// Mitsubishi GX Works2 project: PLC_Group_12   PLC: FX3G

// global labels: Global1
VAR_GLOBAL CONSTANT
  Mixing_Premium_Time : INT := 50;
END_VAR
VAR_GLOBAL
  StartDay AT X007 : BOOL;
  EmergencyStop AT X005 : BOOL;
  LackOfMaterial AT M1 : BOOL;
  DayActive AT M0 : BOOL;
  WorkdayLamp AT Y007 : BOOL;
  RaspberryStock AT D1200 : REAL;
  LemonStock AT D1210 : REAL;
  InitLemon AT D1110 : REAL;
  InitStabilizer AT D1120 : REAL;
  StabilizerStock AT D1220 : REAL;
  BearsStock AT D1230 : REAL;
  InitBears AT D1130 : REAL;
  StorageCount AT D1300 : REAL;
  AnalogOutput AT D8282 : INT;
  StartPreparation AT X001 : BOOL;
  IsPremium AT M3 : BOOL;
  AnalogInput1 AT D8280 : INT;
END_VAR
VAR_GLOBAL CONSTANT
  MinRaspberryPremium : REAL := 385;
  MinLemonPremium : REAL := 665;
  MinStabilizerPremium : REAL := 210;
  MinBearsPremium : REAL := 70;
END_VAR
VAR_GLOBAL
  PreparationActive AT M5 : BOOL;
  IsRegular AT M2 : BOOL;
END_VAR
VAR_GLOBAL CONSTANT
  MinRaspberryRegular : REAL;
  MinBearsRegular : REAL := 28;
  MinStabilizerRegular : REAL := 105;
END_VAR
VAR_GLOBAL
  PreparationLamp AT Y000 : BOOL;
END_VAR
VAR_GLOBAL CONSTANT
  PrepTime : INT := 50;
END_VAR
VAR_GLOBAL
  PreparationDone AT M10 : BOOL;
  CoolingActive AT M7 : BOOL;
  CoolingDone AT M8 : BOOL;
  StartCooling AT X002 : BOOL;
  CoolingLamp AT Y002 : BOOL;
  MixingDone AT M42 : BOOL;
  MixingActive AT M41 : BOOL;
END_VAR
VAR_GLOBAL CONSTANT
  MixingPremiumTime : INT := 50;
END_VAR
VAR_GLOBAL
  InitRaspbery AT D1100 : REAL;
END_VAR
VAR_GLOBAL CONSTANT
  MinLemonRegular : REAL := 455;
  MinStabilizer : REAL := 105;
END_VAR
VAR_GLOBAL
  RaspberryOKRegular AT M20 : BOOL;
  LemonOKRegular AT M21 : BOOL;
  StabilizerOKRegular AT M22 : BOOL;
  BearsOkRegular AT M23 : BOOL;
  RaspberryOKPremium AT M30 : BOOL;
  LemonOKPremium AT M31 : BOOL;
  StabilizerOKPremium AT M32 : BOOL;
  BearsOKPremium AT M33 : BOOL;
  MaterialOk AT M1 : BOOL;
END_VAR
VAR_GLOBAL CONSTANT
  MixingRegularTimee : INT := 30;
END_VAR
VAR_GLOBAL
  FloatInput1 AT D1400 : REAL;
  AnalogScaledInput AT D1402 : REAL;
  TC0 AT T0 : BOOL;
  TS0 AT T0 : BOOL;
  RaspberryTank AT D1500 : REAL;
  LemonTank AT D1550 : REAL;
  TooColdTemp AT X003 : BOOL;
  TC1 AT T1 : BOOL;
  TS1 AT T1 : BOOL;
  LemonCoolingT AT D2000 : REAL;
  RaspberryCoolingT AT D2100 : REAL;
  MixingTank AT D3000 : REAL;
  TC2 AT T2 : BOOL;
  TS2 AT T2 : BOOL;
  TC3 AT T3 : BOOL;
  TS3 AT T3 : BOOL;
  TC4 AT T4 : BOOL;
  TS4 AT T4 : BOOL;
  TC5 AT T5 : BOOL;
  TS5 AT T5 : BOOL;
  MixingLed1 AT Y005 : BOOL;
  MixingLed2 AT Y006 : BOOL;
  TotalUnits AT D4000 : REAL;
  Packages AT D7000 : REAL;
  IsPremium1 AT M11 : BOOL;
  IsPremium2 AT M12 : BOOL;
END_VAR

// task Task_01 (event TRUE, interval 0, priority 31): POU_01

PROGRAM POU_01
VAR
  Init_Raspberry : REAL;
  InitRaspberry : BOOL;
END_VAR
(* structured ladder/FBD written out as ST: instructions are called as NAME(EN, inputs, outputs); _pN, _eN, _tN stand for wires *)
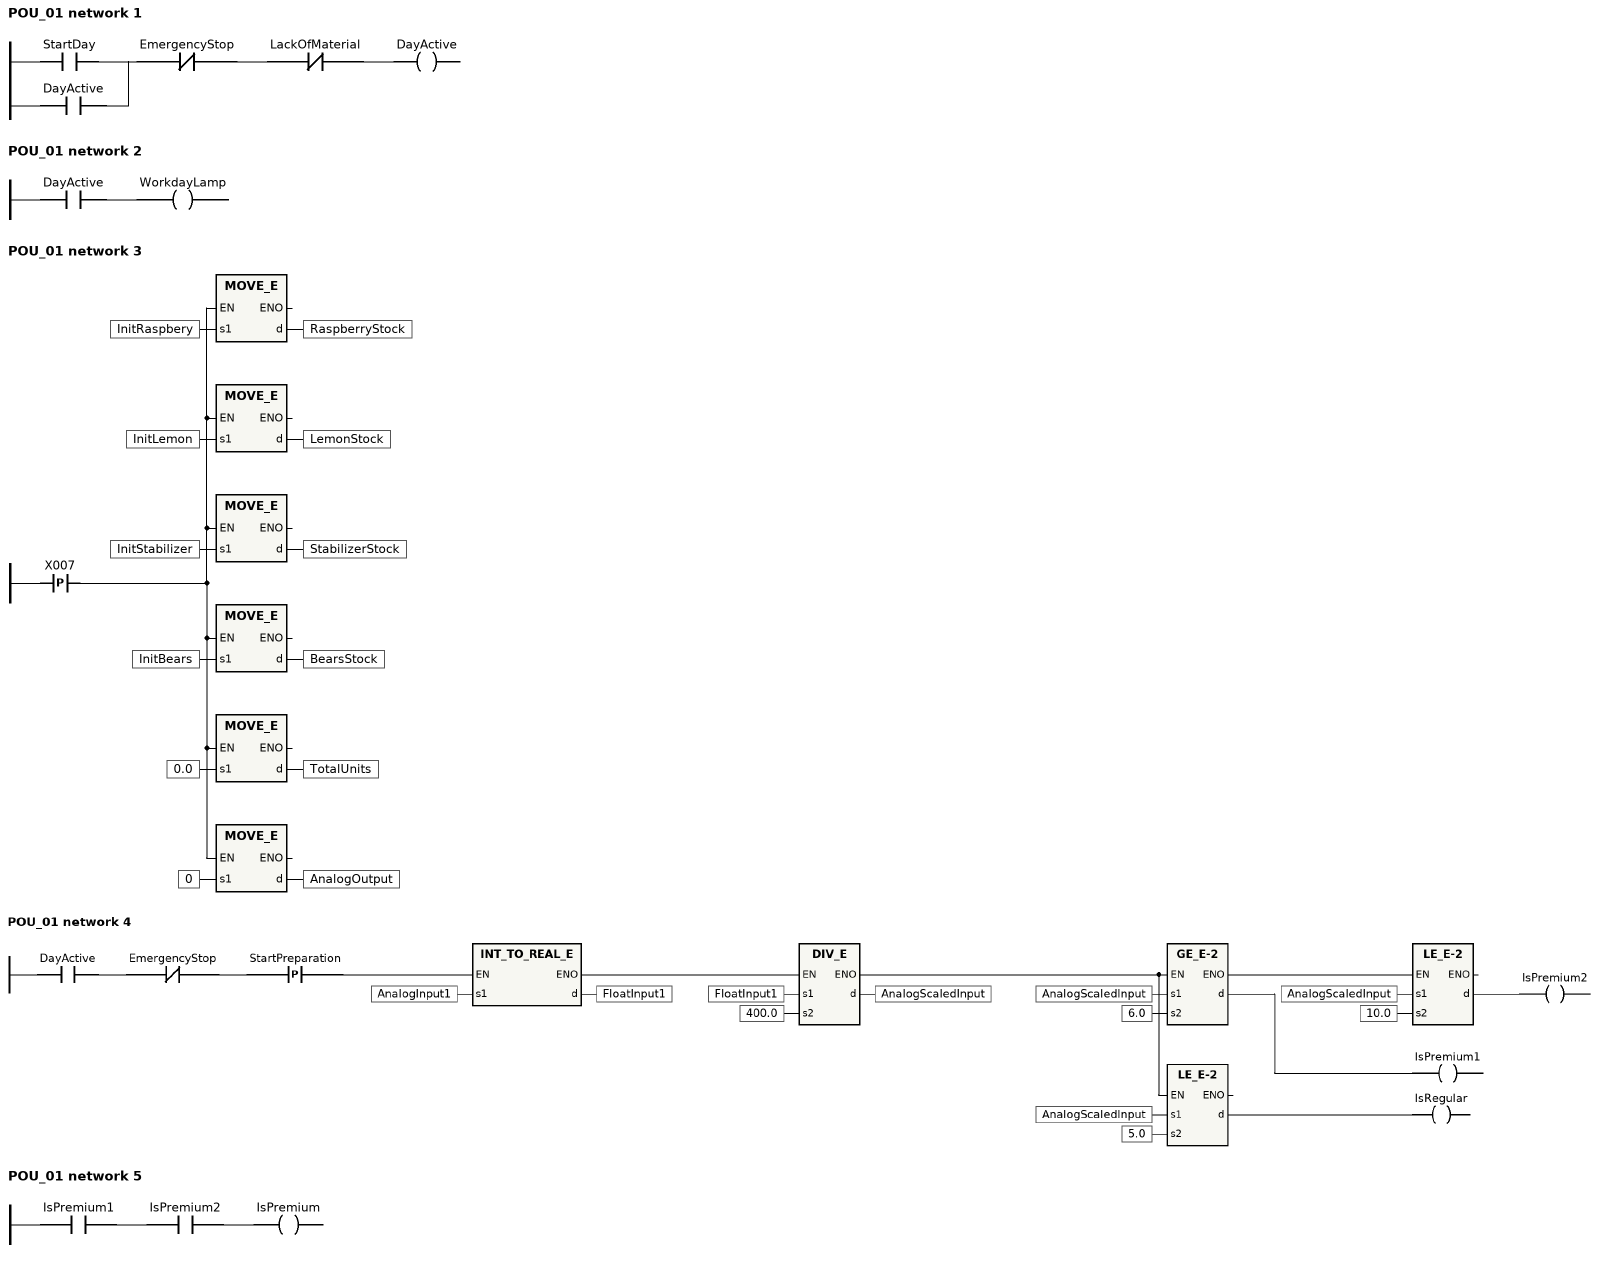
(* network 1 *)
DayActive := ((StartDay OR DayActive) AND NOT EmergencyStop) AND NOT LackOfMaterial;
(* network 2 *)
WorkdayLamp := DayActive;
(* network 3 *)
_p1 := LDP(TRUE, X007);
MOVE_E(_p1, InitRaspbery, RaspberryStock);
MOVE_E(_p1, InitLemon, LemonStock);
MOVE_E(_p1, InitStabilizer, StabilizerStock);
MOVE_E(_p1, InitBears, BearsStock);
MOVE_E(_p1, 0.0, TotalUnits);
MOVE_E(_p1, 0, AnalogOutput);
(* network 4 *)
_e1 := INT_TO_REAL_E(DayActive AND NOT EmergencyStop AND LDP(TRUE, StartPreparation), AnalogInput1, FloatInput1);
_e2 := DIV_E(_e1, FloatInput1, 400.0, AnalogScaledInput);
_e4 := GE_E(_e2, AnalogScaledInput, 6.0, _t3);
LE_E(_e4, AnalogScaledInput, 10.0, _t5);
IsPremium1 := _t3;
IsPremium2 := _t5;
LE_E(_e2, AnalogScaledInput, 5.0, _t6);
IsRegular := _t6;
(* network 5 *)
IsPremium := IsPremium1 AND IsPremium2;
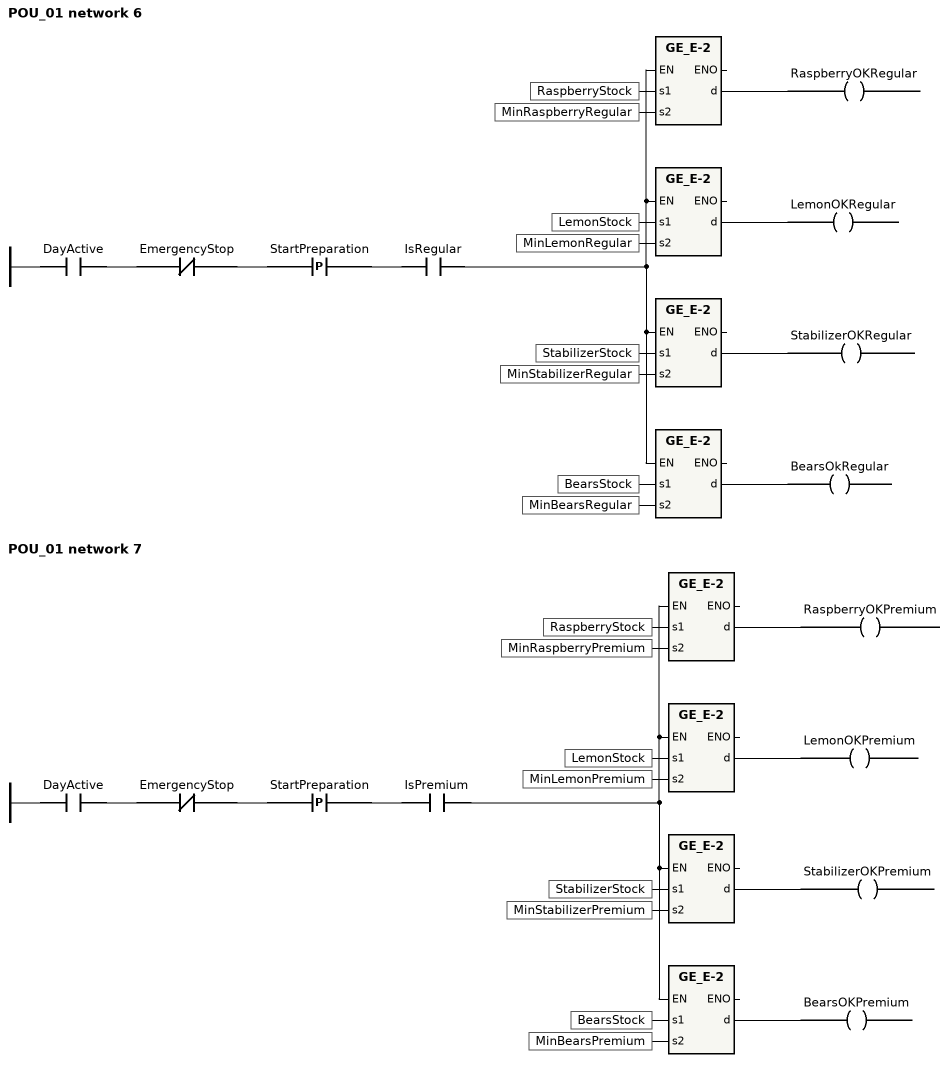
(* network 6 *)
_p1 := DayActive AND NOT EmergencyStop AND LDP(TRUE, StartPreparation) AND IsRegular;
GE_E(_p1, RaspberryStock, MinRaspberryRegular, _t2);
RaspberryOKRegular := _t2;
GE_E(_p1, LemonStock, MinLemonRegular, _t3);
LemonOKRegular := _t3;
GE_E(_p1, StabilizerStock, MinStabilizerRegular, _t4);
StabilizerOKRegular := _t4;
GE_E(_p1, BearsStock, MinBearsRegular, _t5);
BearsOkRegular := _t5;
(* network 7 *)
_p1 := DayActive AND NOT EmergencyStop AND LDP(TRUE, StartPreparation) AND IsPremium;
GE_E(_p1, RaspberryStock, MinRaspberryPremium, _t2);
RaspberryOKPremium := _t2;
GE_E(_p1, LemonStock, MinLemonPremium, _t3);
LemonOKPremium := _t3;
GE_E(_p1, StabilizerStock, MinStabilizerPremium, _t4);
StabilizerOKPremium := _t4;
GE_E(_p1, BearsStock, MinBearsPremium, _t5);
BearsOKPremium := _t5;
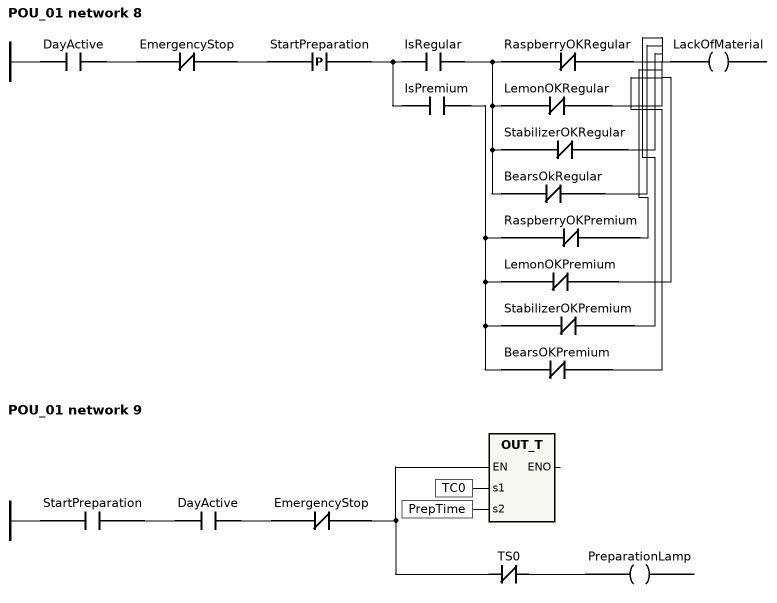
(* network 8 *)
_p1 := DayActive AND NOT EmergencyStop AND LDP(TRUE, StartPreparation);
_p2 := _p1 AND IsRegular;
_p3 := _p1 AND IsPremium;
LackOfMaterial := (_p2 AND NOT RaspberryOKRegular) OR (_p2 AND NOT LemonOKRegular) OR (_p2 AND NOT StabilizerOKRegular) OR (_p2 AND NOT BearsOkRegular) OR (_p3 AND NOT RaspberryOKPremium) OR (_p3 AND NOT LemonOKPremium) OR (_p3 AND NOT StabilizerOKPremium) OR (_p3 AND NOT BearsOKPremium);
(* network 9 *)
_p1 := StartPreparation AND DayActive AND NOT EmergencyStop;
OUT_T(_p1, TC0, PrepTime);
PreparationLamp := _p1 AND NOT TS0;
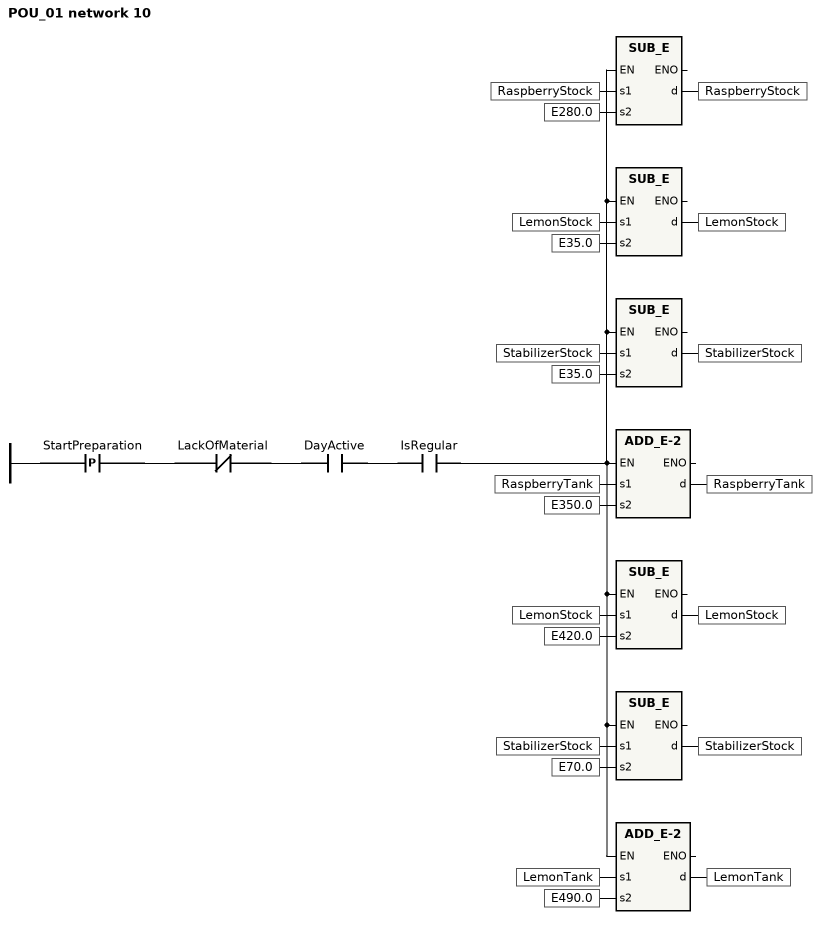
(* network 10 *)
_p1 := LDP(TRUE, StartPreparation) AND NOT LackOfMaterial AND DayActive AND IsRegular;
SUB_E(_p1, RaspberryStock, E280.0, RaspberryStock);
SUB_E(_p1, LemonStock, E35.0, LemonStock);
SUB_E(_p1, StabilizerStock, E35.0, StabilizerStock);
ADD_E(_p1, RaspberryTank, E350.0, RaspberryTank);
SUB_E(_p1, LemonStock, E420.0, LemonStock);
SUB_E(_p1, StabilizerStock, E70.0, StabilizerStock);
ADD_E(_p1, LemonTank, E490.0, LemonTank);
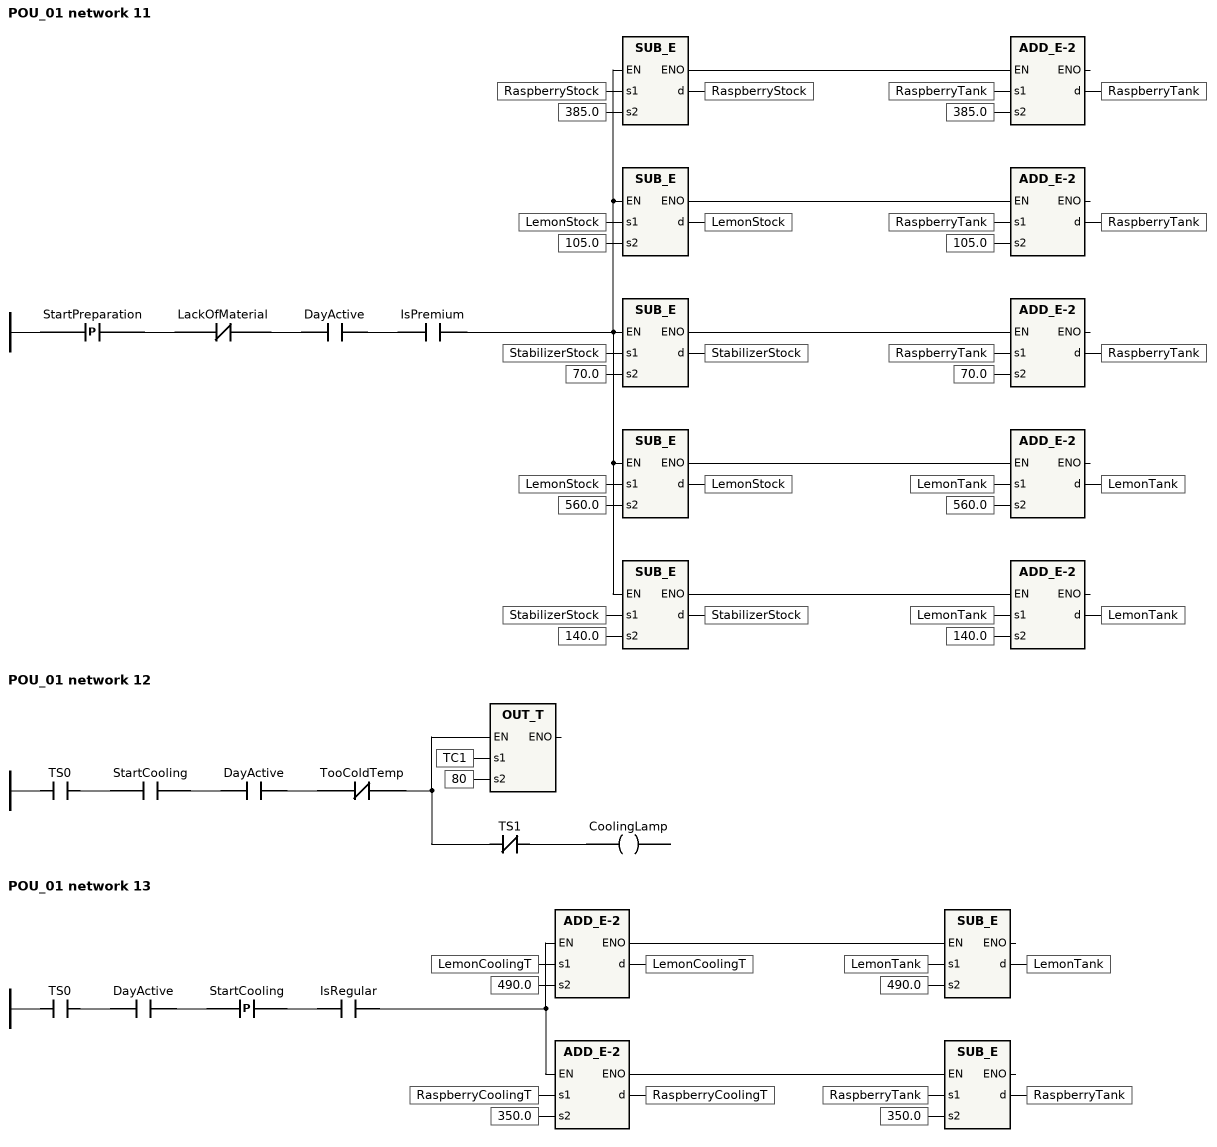
(* network 11 *)
_p1 := LDP(TRUE, StartPreparation) AND NOT LackOfMaterial AND DayActive AND IsPremium;
_e2 := SUB_E(_p1, RaspberryStock, 385.0, RaspberryStock);
ADD_E(_e2, RaspberryTank, 385.0, RaspberryTank);
_e3 := SUB_E(_p1, LemonStock, 105.0, LemonStock);
ADD_E(_e3, RaspberryTank, 105.0, RaspberryTank);
_e4 := SUB_E(_p1, StabilizerStock, 70.0, StabilizerStock);
ADD_E(_e4, RaspberryTank, 70.0, RaspberryTank);
_e5 := SUB_E(_p1, LemonStock, 560.0, LemonStock);
ADD_E(_e5, LemonTank, 560.0, LemonTank);
_e6 := SUB_E(_p1, StabilizerStock, 140.0, StabilizerStock);
ADD_E(_e6, LemonTank, 140.0, LemonTank);
(* network 12 *)
_p1 := TS0 AND StartCooling AND DayActive AND NOT TooColdTemp;
OUT_T(_p1, TC1, 80);
CoolingLamp := _p1 AND NOT TS1;
(* network 13 *)
_p1 := TS0 AND DayActive AND LDP(TRUE, StartCooling) AND IsRegular;
_e2 := ADD_E(_p1, LemonCoolingT, 490.0, LemonCoolingT);
SUB_E(_e2, LemonTank, 490.0, LemonTank);
_e3 := ADD_E(_p1, RaspberryCoolingT, 350.0, RaspberryCoolingT);
SUB_E(_e3, RaspberryTank, 350.0, RaspberryTank);
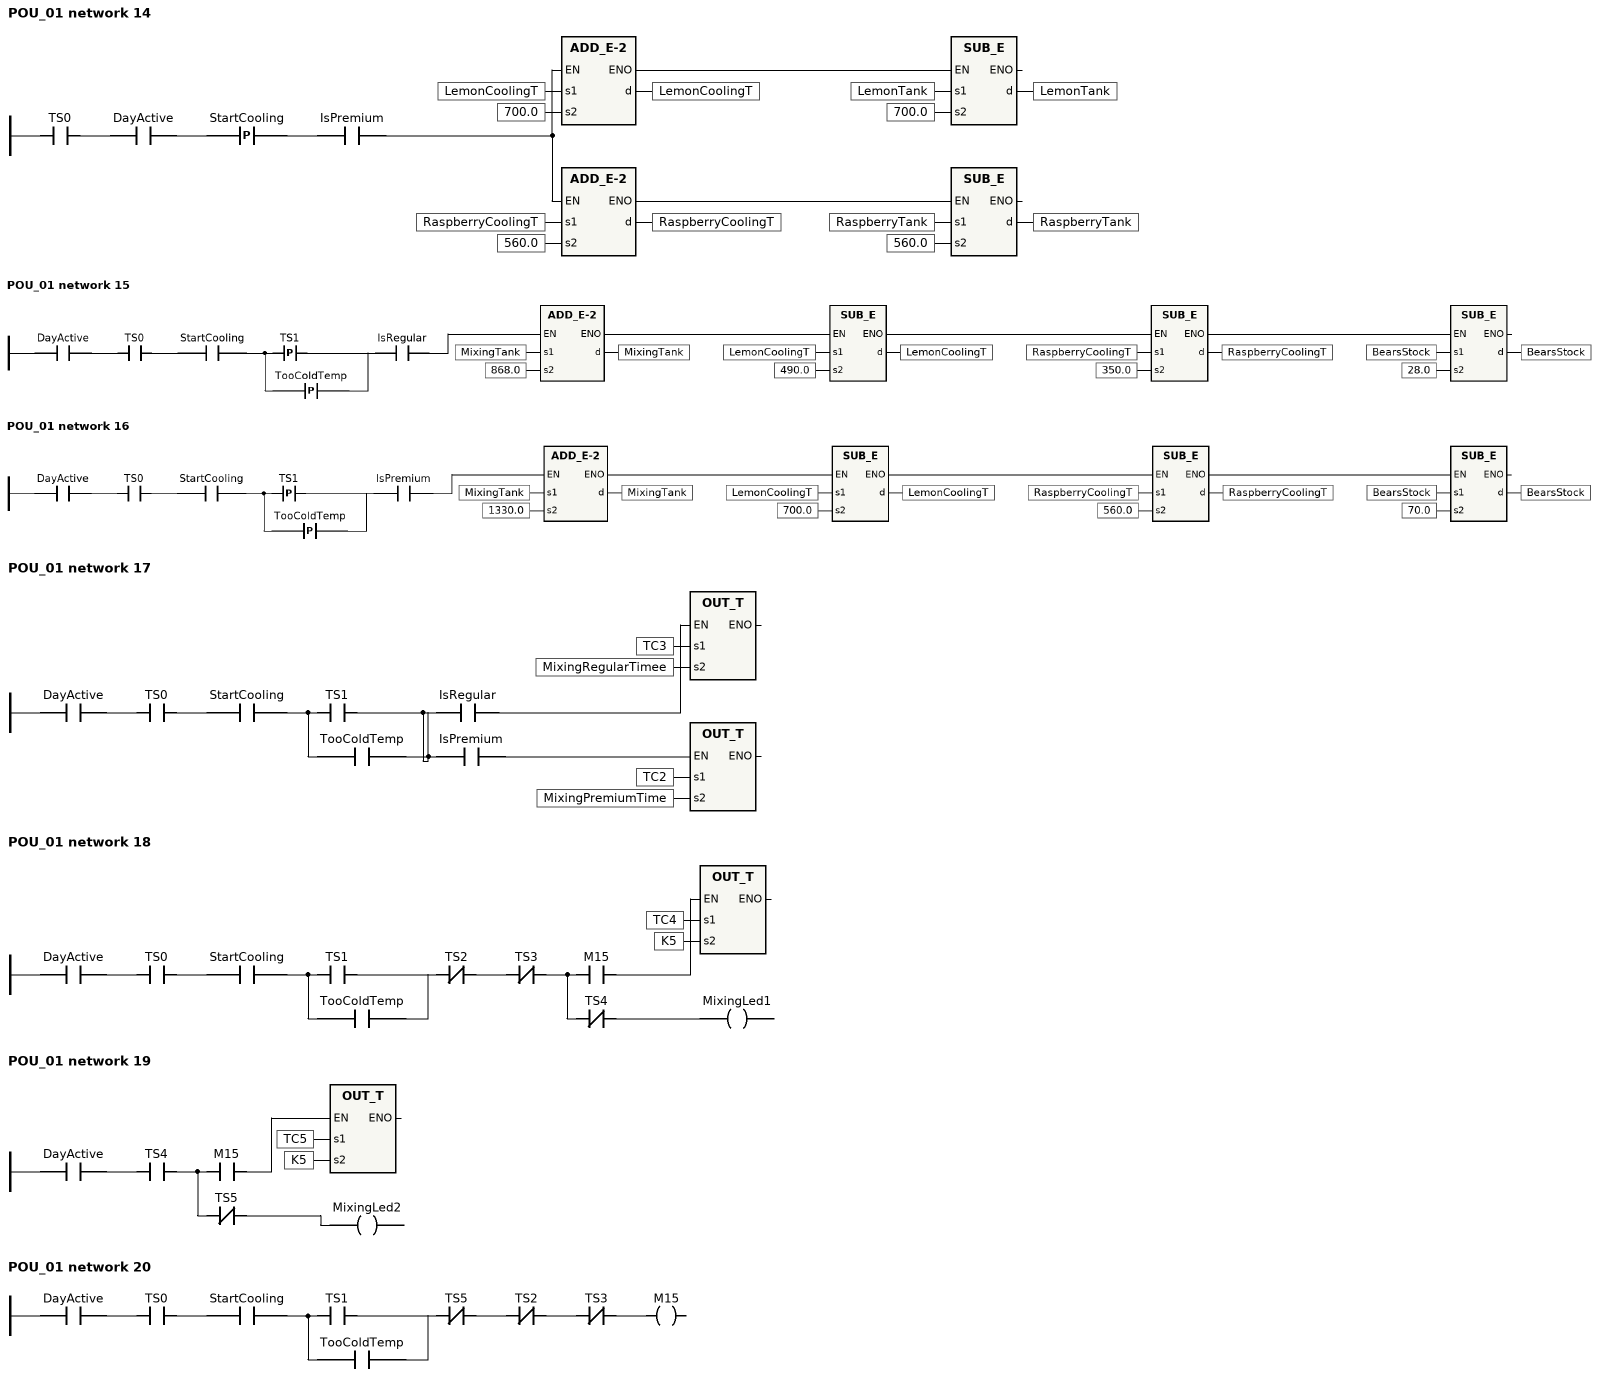
(* network 14 *)
_p1 := TS0 AND DayActive AND LDP(TRUE, StartCooling) AND IsPremium;
_e2 := ADD_E(_p1, LemonCoolingT, 700.0, LemonCoolingT);
SUB_E(_e2, LemonTank, 700.0, LemonTank);
_e3 := ADD_E(_p1, RaspberryCoolingT, 560.0, RaspberryCoolingT);
SUB_E(_e3, RaspberryTank, 560.0, RaspberryTank);
(* network 15 *)
_p1 := DayActive AND TS0 AND StartCooling;
_e2 := ADD_E(((_p1 AND LDP(TRUE, TS1)) OR (_p1 AND LDP(TRUE, TooColdTemp))) AND IsRegular, MixingTank, 868.0, MixingTank);
_e3 := SUB_E(_e2, LemonCoolingT, 490.0, LemonCoolingT);
_e4 := SUB_E(_e3, RaspberryCoolingT, 350.0, RaspberryCoolingT);
SUB_E(_e4, BearsStock, 28.0, BearsStock);
(* network 16 *)
_p1 := DayActive AND TS0 AND StartCooling;
_e2 := ADD_E(((_p1 AND LDP(TRUE, TS1)) OR (_p1 AND LDP(TRUE, TooColdTemp))) AND IsPremium, MixingTank, 1330.0, MixingTank);
_e3 := SUB_E(_e2, LemonCoolingT, 700.0, LemonCoolingT);
_e4 := SUB_E(_e3, RaspberryCoolingT, 560.0, RaspberryCoolingT);
SUB_E(_e4, BearsStock, 70.0, BearsStock);
(* network 17 *)
_p1 := DayActive AND TS0 AND StartCooling;
_p2 := (_p1 AND TS1) OR (_p1 AND TooColdTemp);
OUT_T(_p2 AND IsRegular, TC3, MixingRegularTimee);
OUT_T(_p2 AND IsPremium, TC2, MixingPremiumTime);
(* network 18 *)
_p1 := DayActive AND TS0 AND StartCooling;
_p2 := (((_p1 AND TS1) OR (_p1 AND TooColdTemp)) AND NOT TS2) AND NOT TS3;
OUT_T(_p2 AND M15, TC4, K5);
MixingLed1 := _p2 AND NOT TS4;
(* network 19 *)
_p1 := DayActive AND TS4;
OUT_T(_p1 AND M15, TC5, K5);
MixingLed2 := _p1 AND NOT TS5;
(* network 20 *)
_p1 := DayActive AND TS0 AND StartCooling;
M15 := ((((_p1 AND TS1) OR (_p1 AND TooColdTemp)) AND NOT TS5) AND NOT TS2) AND NOT TS3;
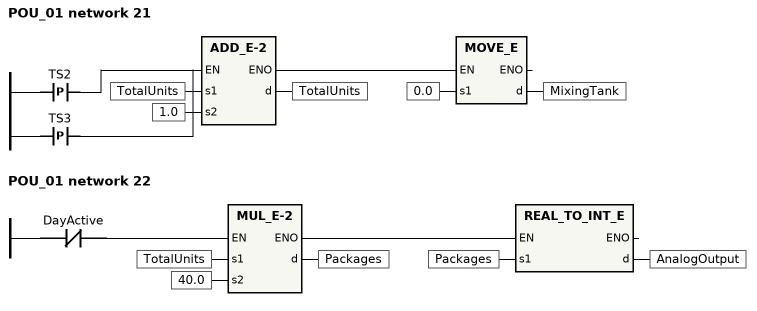
(* network 21 *)
_e1 := ADD_E(LDP(TRUE, TS2) OR LDP(TRUE, TS3), TotalUnits, 1.0, TotalUnits);
MOVE_E(_e1, 0.0, MixingTank);
(* network 22 *)
_e1 := MUL_E(NOT DayActive, TotalUnits, 40.0, Packages);
REAL_TO_INT_E(_e1, Packages, AnalogOutput);
END_PROGRAM
